// TwinCAT 3 PLC project Test
// ProgramVersion: 3.1.4023.0
// libraries:
//   Tc2_Standard, * (Beckhoff Automation GmbH)
//   Tc2_System, * (Beckhoff Automation GmbH)
//   Tc2_Utilities, * (Beckhoff Automation GmbH)
//   Tc3_Module, * (Beckhoff Automation GmbH)
// project tree:
//   DUTs/ Access_levels.TcDUT, dut_Setting.TcDUT, S_Drive_control_settings.TcDUT, S_General_settings.TcDUT, S_TPD32_base_settings.TcDUT
//   GVLs/ Gen.TcGVL, SpeedGuardian.TcGVL, sp.TcGVL, spHMI.TcGVL, Torque_prediction.TcGVL, tst.TcGVL
//   / PlcTask.TcTTO
//   POUs/ FB_DateTime.TcPOU, FB_Moving_average.TcPOU, FB_Torque_prediction.TcPOU, MAIN.TcPOU
// real-time tasks:
//   TASK PlcTask: cycle T#1ms, priority 20, ADS port 350

CONFIGURATION Test
    RESOURCE PLC ON TwinCAT3
        TASK PlcTask(INTERVAL := T#1ms, PRIORITY := 20);
        PROGRAM MAIN WITH PlcTask : MAIN;
    END_RESOURCE
END_CONFIGURATION

// ---- DUTs/Access_levels.TcDUT
{attribute 'qualified_only'}
{attribute 'strict'}
TYPE Access_levels :
(
	Driver := 0,
	Electrician := 1,
	Foreman := 2,
	Engineer := 3,
	Admin := 4
);
END_TYPE

// ---- DUTs/dut_Setting.TcDUT
TYPE dut_Setting :
STRUCT
	Val: REAL;
	Desc: STRING;
	Unit: STRING;
	Minimum: REAL;
	Maximum: REAL;
	Write_level:REAL;
END_STRUCT
END_TYPE

// ---- DUTs/S_Drive_control_settings.TcDUT
TYPE S_Drive_control_settings :
STRUCT
	Max_drive_speed:dut_Setting := (Val:=0,Desc:='Maximum drive speed',Unit:='m/s',Minimum:=0,Maximum:=7);
	Max_drive_torque:dut_Setting := (Val:=0,Desc:='Maximum drive torque',Unit:='m/s',Minimum:=0,Maximum:=7);
	Speed_S_func_scans:dut_Setting := (Val:=0,Desc:='Speed S function scans',Unit:='m/s',Minimum:=0,Maximum:=7);
	Current_S_func_scans:dut_Setting := (Val:=0,Desc:='Current S function scans',Unit:='m/s',Minimum:=0,Maximum:=7);
	No_start_time:dut_Setting := (Val:=0,Desc:='No-start time',Unit:='m/s',Minimum:=0,Maximum:=7);
	Motor_fed_delay:dut_Setting := (Val:=0,Desc:='Motor fed delay',Unit:='m/s',Minimum:=0,Maximum:=7);
	Stall_time:dut_Setting := (Val:=0,Desc:='Stall time',Unit:='m/s',Minimum:=0,Maximum:=7);
	Stall_speed:dut_Setting := (Val:=0,Desc:='Stall speed',Unit:='m/s',Minimum:=0,Maximum:=7);
	Torque_ctrl_max_speed:dut_Setting := (Val:=0,Desc:='Torque control maximum speed',Unit:='m/s',Minimum:=0,Maximum:=7);
	Brake_apply_speed:dut_Setting := (Val:=0,Desc:='Brake apply speed',Unit:='m/s',Minimum:=0,Maximum:=7);
	Trail_brake_speed:dut_Setting := (Val:=0,Desc:='Trail brake speed',Unit:='m/s',Minimum:=0,Maximum:=7);
	De_energise_to_trail:BOOL;
	Single_lever_control:BOOL;
	Stall_current:dut_Setting := (Val:=0,Desc:='Stall current',Unit:='m/s',Minimum:=0,Maximum:=7);
	Backout_min_speed:dut_Setting := (Val:=0,Desc:='Backout minimum speed',Unit:='m/s',Minimum:=0,Maximum:=7);

	(*Torque prediction settings*)	
	Lh_cage_mass_current:dut_Setting := (Val:=0,Desc:='Left-hand cage mass current',Unit:='m/s',Minimum:=0,Maximum:=7);
	Rh_cage_mass_current:dut_Setting := (Val:=0,Desc:='Right-hand cage mass current',Unit:='m/s',Minimum:=0,Maximum:=7);
	Lh_rope_mass_current:dut_Setting := (Val:=0,Desc:='Left-hand rope mass current',Unit:='m/s',Minimum:=0,Maximum:=7);
	Rh_rope_mass_current:dut_Setting := (Val:=0,Desc:='Right-hand rope mass current',Unit:='m/s',Minimum:=0,Maximum:=7);
	Full_payload_current:dut_Setting := (Val:=0,Desc:='Full payload current',Unit:='m/s',Minimum:=0,Maximum:=7);
	A_s2_per_m:dut_Setting := (Val:=0,Desc:='A S2 per meter',Unit:='m/s',Minimum:=0,Maximum:=7);
	Accel_torque_lag:dut_Setting := (Val:=0,Desc:='Accelleration torque lag',Unit:='m/s',Minimum:=0,Maximum:=7);
	Dynamic_friction_current:dut_Setting := (Val:=0,Desc:='Dynamic friction current',Unit:='m/s',Minimum:=0,Maximum:=7);

END_STRUCT
END_TYPE

// ---- DUTs/S_General_settings.TcDUT
TYPE S_General_settings :
STRUCT
	Full_speed: dut_Setting := (Val:=0,Desc:='Full Speed',Unit:='m/s',Minimum:=0,Maximum:=7);
	Slow_switch_speed: dut_Setting  := (Val:=0,Desc:='Slow switch speed',Unit:='m/s',Minimum:=0,Maximum:=7);
END_STRUCT
END_TYPE

// ---- DUTs/S_TPD32_base_settings.TcDUT
TYPE S_TPD32_base_settings :
STRUCT
	Motor_base_rpm:dut_Setting := (Val:=0,Desc:='Rated rpm of the motor',Unit:='m/s',Minimum:=0,Maximum:=7); (*Rated rpm of the motor*)
	Max_output_voltage:dut_Setting := (Val:=0,Desc:='Maximum DC armature voltage',Unit:='m/s',Minimum:=0,Maximum:=7); (*Maximum DC armature voltage*)
	Full_load_curr:dut_Setting := (Val:=0,Desc:='Rated armature amps of the motor',Unit:='m/s',Minimum:=0,Maximum:=7); (*Rated armature amps of the motor*)
	DCV_nominal_flux_current:dut_Setting := (Val:=0,Desc:='Nominal flux current of the DCV according to S14 DIP switches',Unit:='m/s',Minimum:=0,Maximum:=7); (*Nominal flux current of the DCV according to S14 DIP switches*)
	Motor_nominal_flux_current:dut_Setting := (Val:=0,Desc:='Nominal flux current of the DCV according to S14 DIP switches',Unit:='m/s',Minimum:=0,Maximum:=7); (*Nominal flux current of the DCV according to S14 DIP switches*)
	Flux_current_min:dut_Setting := (Val:=0,Desc:='Percentage of rated motor field current for field weakening',Unit:='m/s',Minimum:=0,Maximum:=7); (*Percentage of rated motor field current for field weakening*)
	Acc_delta_time:dut_Setting := (Val:=0,Desc:='Acceleration time from zero to rated motor rpm in seconds',Unit:='m/s',Minimum:=0,Maximum:=7); (*Acceleration time from zero to rated motor rpm in seconds*)
	Dec_delta_time:dut_Setting := (Val:=0,Desc:='Deceleration time from rated motor rpm to zero in seconds',Unit:='m/s',Minimum:=0,Maximum:=7); (*Deceleration time from rated motor rpm to zero in seconds*)
END_STRUCT
END_TYPE

// ---- GVLs/Gen.TcGVL
{attribute 'qualified_only'}
VAR_GLOBAL
	DateTime: DATE_AND_TIME;
	
	Lh_depth: REAL;
	Rh_depth: REAL;
	Lh_speed: REAL;
	Rh_speed: REAL;
	
	Rh_up: BOOL;
END_VAR

// ---- GVLs/SpeedGuardian.TcGVL
{attribute 'qualified_only'}
VAR_GLOBAL
		Lh_overwind: BOOL;
		Lh_underwind: BOOL;
		Rh_overwind: BOOL;
		Rh_underwind: BOOL;
END_VAR

// ---- GVLs/sp.TcGVL
{attribute 'qualified_only'}
VAR_GLOBAL
	Gen: S_General_settings;
	Drive: S_Drive_control_settings;
	TPD: S_TPD32_base_settings;
END_VAR

// ---- GVLs/spHMI.TcGVL
{attribute 'qualified_only'}
VAR_GLOBAL
	Gen: S_General_settings;
	Drive: S_Drive_control_settings;
	TPD: S_TPD32_base_settings;
END_VAR

// ---- GVLs/Torque_prediction.TcGVL
{attribute 'qualified_only'}
VAR_GLOBAL
	On: BOOL;
	Set: BOOL;
	Reset: BOOL;
	
	Lh_full: BOOL;
	Lh_half: BOOL;
	Equal: BOOL;
	Rh_half: BOOL;
	Rh_full: BOOL;
	
	Lh_full_request: BOOL;
	Lh_half_request: BOOL;
	Equal_request: BOOL;
	Rh_half_request: BOOL;
	Rh_full_request: BOOL;
END_VAR

// ---- GVLs/tst.TcGVL
{attribute 'qualified_only'}
VAR_GLOBAL
	testBool1:BOOL := TRUE;
	testStr1:STRING := 'stringy string';
	testReal1:REAL := 1520;
END_VAR

// ---- POUs/MAIN.TcPOU
PROGRAM MAIN
VAR
	TP0: FB_Torque_prediction;	
	MA0: FB_Moving_average;
	
	X: REAL:= 0;
	Y: REAL;
		
	sDateTime: STRING;
	FB_DateTime_0: FB_DateTime;
	i: INT;
	Full_speed: REAL:= 5;
	Creep_speed: REAL:= 0.5;
	Creep_in_dist: REAL:= 5.0;
	Creep_out_dist: REAL:= 2.0;
	Accel: REAL:= 0.7;
	Distance: REAL;
	Bottom_depth: REAL:= 100;
END_VAR

VAR_OUTPUT
	Allowed_speed: REAL;
	Prev_depth: REAL;
	Restriction: REAL;
END_VAR

TP0();
FB_DateTime_0(sDateTime => sDateTime);

MA0(New_sample:= X, Num_samples:= 201, Out=> Y);
X:= X + 1;
IF X > 200 + 0.1 THEN
	X:= 0.0;
END_IF

FOR i := 1 TO 10000 DO
	Allowed_speed:= SQRT(Creep_speed*Creep_speed + 2*Accel*Distance);
END_FOR

Gen.Rh_depth:= Gen.Rh_depth + Gen.Rh_speed/1000;
	
IF Gen.Rh_up THEN
	Allowed_speed:= Full_speed;	
	IF Gen.Rh_depth < Creep_in_dist THEN
		Allowed_speed:= Creep_speed;
	ELSE	
		Restriction:= SQRT(Creep_speed*Creep_speed + 2*Accel*(Gen.Rh_depth - Creep_in_dist));
		IF Restriction < Allowed_speed THEN
			Allowed_speed:= Restriction;
		END_IF;	
	END_IF;
	
	IF Gen.Rh_depth > Bottom_depth - Creep_out_dist THEN
		Allowed_speed:= Creep_speed;
	ELSE	
		Restriction:= SQRT(Creep_speed*Creep_speed + 2*Accel*(Bottom_depth - Gen.Rh_depth + Creep_out_dist));
		IF Restriction < Allowed_speed THEN
			Allowed_speed:= Restriction;
		END_IF;	
	END_IF;
	
	IF Gen.Rh_depth < 0 THEN
		Gen.Rh_depth:= 0;
		Gen.Rh_up := FALSE;
	END_IF
	Gen.Rh_speed:= -Allowed_speed;
ELSE
	Allowed_speed:= Full_speed;	
	IF Gen.Rh_depth < Creep_out_dist THEN
		Allowed_speed:= Creep_speed;
	ELSE	
		Restriction:= SQRT(Creep_speed*Creep_speed + 2*Accel*(Gen.Rh_depth - Creep_out_dist));
		IF Restriction < Allowed_speed THEN
			Allowed_speed:= Restriction;
		END_IF;	
	END_IF;
	
	IF Gen.Rh_depth > Bottom_depth - Creep_in_dist THEN
		Allowed_speed:= Creep_speed;
	ELSE	
		Restriction:= SQRT(Creep_speed*Creep_speed + 2*Accel*(Bottom_depth - Gen.Rh_depth + Creep_in_dist));
		IF Restriction < Allowed_speed THEN
			Allowed_speed:= Restriction;
		END_IF;	
	END_IF;
	
	IF Gen.Rh_depth < 0 THEN
		Gen.Rh_depth:= 0;
		Gen.Rh_up := FALSE;
	END_IF

	IF Gen.Rh_depth > Bottom_depth THEN
		Gen.Rh_depth:= Bottom_depth;
		Gen.Rh_up := TRUE;
	END_IF
	Gen.Rh_speed:= Allowed_speed;
END_IF

Gen.Lh_depth:= Bottom_depth - Gen.Rh_depth;
Gen.Lh_speed:= -Gen.Rh_speed;

END_PROGRAM

// ---- POUs/FB_Torque_prediction.TcPOU
FUNCTION_BLOCK FB_Torque_prediction
VAR_INPUT
END_VAR
VAR_OUTPUT
END_VAR
VAR
	Lh_full: BOOL;
	Lh_half: BOOL;
	Equal: BOOL;
	Rh_half: BOOL;
	Rh_full: BOOL;
	
	Lh_full_selected: BOOL;
	Lh_half_selected: BOOL;
	Equal_selected: BOOL;
	Rh_half_selected: BOOL;
	Rh_full_selected: BOOL;
	
	R_TRIG0: R_TRIG;
	R_TRIG1: R_TRIG;
	R_TRIG2: R_TRIG;
	R_TRIG3: R_TRIG;
	R_TRIG4: R_TRIG;
END_VAR

R_TRIG0(CLK:= Torque_prediction.Lh_full_request, Q=> Lh_full_selected);
R_TRIG1(CLK:= Torque_prediction.Lh_half_request, Q=> Lh_half_selected);
R_TRIG2(CLK:= Torque_prediction.Equal_request, Q=> Equal_selected);
R_TRIG3(CLK:= Torque_prediction.Rh_half_request, Q=> Rh_half_selected);
R_TRIG4(CLK:= Torque_prediction.Rh_full_request, Q=> Rh_full_selected);

IF Lh_full_selected THEN
	Torque_prediction.Lh_full := 1;
	Torque_prediction.Lh_half := 0;
	Torque_prediction.Rh_half := 0;
	Torque_prediction.Rh_full := 0;
ELSIF Lh_half_selected THEN
	Torque_prediction.Lh_full := 0;
	Torque_prediction.Lh_half := 1;
	Torque_prediction.Rh_half := 0;
	Torque_prediction.Rh_full := 0;
ELSIF Equal_selected THEN
	Torque_prediction.Lh_full := 0;
	Torque_prediction.Lh_half := 0;
	Torque_prediction.Rh_half := 0;
	Torque_prediction.Rh_full := 0;
ELSIF Rh_half_selected THEN
	Torque_prediction.Lh_full := 0;
	Torque_prediction.Lh_half := 0;
	Torque_prediction.Rh_half := 1;
	Torque_prediction.Rh_full := 0;
ELSIF Rh_full_selected THEN
	Torque_prediction.Lh_full := 0;
	Torque_prediction.Lh_half := 0;
	Torque_prediction.Rh_half := 0;
	Torque_prediction.Rh_full := 1;
END_IF

Torque_prediction.Equal:= 
	NOT Torque_prediction.Lh_full AND 
	NOT Torque_prediction.Lh_half AND 
	NOT Torque_prediction.Rh_half AND 
	NOT Torque_prediction.Rh_full;

Torque_prediction.Lh_full_request := 0;
Torque_prediction.Lh_half_request := 0;
Torque_prediction.Equal_request := 0;
Torque_prediction.Rh_half_request := 0;
Torque_prediction.Rh_full_request := 0;

IF Torque_prediction.Set THEN
	Torque_prediction.On:= 1;
END_IF
IF Torque_prediction.Reset THEN
	Torque_prediction.On:= 0;
END_IF

END_FUNCTION_BLOCK

// ---- POUs/FB_Moving_average.TcPOU
FUNCTION_BLOCK FB_Moving_average
VAR_INPUT
	New_sample: REAL;
	Num_samples: INT;
END_VAR
VAR_OUTPUT
	Out: REAL;
END_VAR
VAR CONSTANT
	Array_size: INT := 300;	
END_VAR
VAR
	Samples: ARRAY[0..(Array_size - 1)] OF REAL;
	i: INT;
	Sum: REAL;
	Pulse: BOOL;
	Toggle: BOOL;
END_VAR

(* Shift all the array elements one position and add them up while doing so *)
Sum:= 0;
FOR i:= 1 TO Num_samples - 1 DO
	Samples[Num_samples - i]:= Samples[Num_samples - i - 1];
	Sum:= Sum + Samples[Num_samples - i];
END_FOR

(* Insert the new sample into the array and add it to the sum *)
Samples[0]:= New_sample;
Sum:= Sum + New_sample;

(* Calculate the average *)
Out:= Sum / INT_TO_REAL(Num_samples);

END_FUNCTION_BLOCK

// ---- POUs/FB_DateTime.TcPOU
FUNCTION_BLOCK FB_DateTime
VAR_INPUT
END_VAR
VAR_OUTPUT
	sDateTime: STRING;
END_VAR
VAR
	fbTime   : FB_LocalSystemTime := ( bEnable := TRUE, dwCycle := 1 );
	//fbSystemTimeToDT: SYSTEMTIME_TO_DT;
	sTime, sSystemTime, sDate, sMonth, sTemp: STRING;
END_VAR

fbTime();
Gen.DateTime:= SYSTEMTIME_TO_DT(fbTime.systemTime); 

sSystemTime:= SYSTEMTIME_TO_STRING(fbTime.systemTime);

sTime:= RIGHT(CONCAT('0', WORD_TO_STRING(fbTime.systemTime.wHour)), 2);
sTime:= CONCAT(sTime, ':');
sTemp:= CONCAT('0', WORD_TO_STRING(fbTime.systemTime.wMinute));
sTime:= CONCAT(sTime, RIGHT(sTemp, 2));
sTime:= CONCAT(sTime, ':');
sTemp:= CONCAT('0', WORD_TO_STRING(fbTime.systemTime.wSecond));
sTime:= CONCAT(sTime, RIGHT(sTemp, 2));

sDate:= WORD_TO_STRING(fbTime.systemTime.wDay);
sDate:= CONCAT(sDate, ' ');
CASE fbTime.systemTime.wMonth OF
	1: sMonth:= 'January';
	2: sMonth:= 'Febuary';
	3: sMonth:= 'March';
	4: sMonth:= 'April';
	5: sMonth:= 'May';
	6: sMonth:= 'June';
	7: sMonth:= 'July';
	8: sMonth:= 'August';
	9: sMonth:= 'September';
	10: sMonth:= 'October';
	11: sMonth:= 'November';
	12: sMonth:= 'December';
ELSE
	sMonth:= 'Invalid';
END_CASE
sDate:= CONCAT(sDate, sMonth);
sDate:= CONCAT(sDate, ' ');
sDate:= CONCAT(sDate, WORD_TO_STRING(fbTime.systemTime.wYear));

sDateTime:= CONCAT(sDate, CONCAT('\n', sTime));

END_FUNCTION_BLOCK
